PROGRAM PRG_INJ
VAR
END_VAR


// Valves
VCN_70(i_xExtIlkOK:= , i_ReqPos:= , iq_stVCN=> );
//VGP_80
VVC_71(i_xExtILK_OK:= VVC_72.M_IsClosed(), i_xOverrideMode:= , iq_stValve=> );
VVC_72(i_xExtILK_OK:= VVC_71.M_IsClosed(), i_xOverrideMode:= , iq_stValve=> );

//Gauges
GCM_70(VG=> , i_rFULL_SCALE:= 2000);
GCM_80(VG=> , i_rFULL_SCALE:= 20);
GCM_81(VG=> , i_rFULL_SCALE:= 0.25);

END_PROGRAM

(* stored: Version 1.1.0.1, ProductVersion 3.1.4022.12
   POU PRG_INJ: Id {8b858f89-a705-4da6-a8c0-4cd0b412d38f}, SpecialFunc None *)
